TEXTLIST StationName
  0 = '接驳上料' | Chinese: '接驳上料' | English: 'AcquireLoad'
  1 = '转向站' | Chinese: '转向站' | English: 'Steering'
  2 = '解锁站' | Chinese: '解锁站' | English: 'OpenLock'
  3 = '取UC站' | Chinese: '取UC站' | English: 'TakeUc'
  4 = '取Uc模组' | Chinese: '取Uc模组' | English: 'TakeUc_M'
  5 = '下工装站' | Chinese: '下工装站' | English: 'UnloadFrock'
  6 = '下料皮带线' | Chinese: '下料皮带线' | English: 'Unload_L'
  7 = '其他' | Chinese: '其他' | English: 'Other'
   = ''
END_TEXTLIST

(* stored: Version 1.1.0.1, ProductVersion 3.1.4024.3
   TextList StationName: Id {9a8a1e43-7121-4581-9c4a-1d71fa957470} *)
